FUNCTION "CWA_ScaleRead" : VOID	// FC 42
TITLE = CWA READ SCALE
//
//COPYRIGHT:    (C) 1996 BY  BUHLER LTD.
//                           CH-9240 UZWIL  SWITZERLAND
//
//PRODUCT:      CWA
//
//TITLE:        SCALE CONTROL: READ SCALE
//
//-------------------------------------------------------------------------
//
//IDENT:        AUTOR:              DEPT:                         DATE:
//
//FC42.3.1      A. Egli             CT3                           29-Jun-2004
//              InLocal to disable alarm EsReading
//FC42.3.0      A. Egli             CT3                            8-Feb-2000
//              BCD: Check niybble in range '0' to '9'
//FC42.2A       A. Egli             CT3                           23-Feb-99
//              ERG2: DBX125.7: ParErg2Parallel (16+4Bit)
//              Attention: By Pulse input Bit-Number new on DBB134 not DBB135
//FC42.1D       A. Egli             CT3                           22-Oct-98
//              ERG2: DBX125.6: ParErg2DP
//
//FC42.1C       A. Egli             CT3                           16-Jan-98
//              Fault Reading BCD Value
//
//FC42.1B       A. Egli             CT3                           20-Jan-98
//              Update to  Version S5 2A
//
//FC42.1A       S. Kalberer         AEE61                         24-APR-96
//              1st Release in S7, converted from FB42.1B
//
//-------------------------------------------------------------------------
//
//PURPOSE:      MANUAL : CWAMAN
//
//RESTRICTIONS:
//
//-------------------------------------------------------------------------
//
//
//ACTUAL DB BY CALL: SCALE    DB
//
AUTHOR : EA
FAMILY : CWA
NAME : CWARead
VERSION : 3.1
VAR_TEMP
  AddrPointer : DWORD ;
  tmpValue : DWORD ;
END_VAR
BEGIN
NETWORK
TITLE = BCD/ERG
      AN    DBX 125.1;	// ParERG
      AN    DBX 125.0;	// ParBCD
      JC    NX02;
      A     DBX 57.0;	// inp_ReadingLocked
      O     DBX 125.5;	// ParmeasurmentASW
      JC    NX02;
      A     DBX 125.1;	// ParERG
      JC    ERG;	// === BCD (MINIPOND)==============
      L     DBB 135;	// ParAddrInp2Word
      SLD   3;
      T     #AddrPointer;
      L     DBB 134;	// ParAddrInpBit
      L     PIW [#AddrPointer];	// temp2
      SRW;	// Bit 0= sign
      T     DBW 154;	// --> temp2
      AN    DBX 155.1;	// inp_data_ready
      JC    D_R;
      L     DBW 132;	// ParAddrInp1Word
      SLD   3;
      T     #AddrPointer;
      L     PIW [#AddrPointer];
      T     DBW 152;	// --> temp1
      L     W#16#FFFF;
      ==I;
      JC    ERR1;	// --> reading error
// Begin [3A]  
//    Tesat Digit in range ['0' .. '9']   
      L     DBW 152;	// temp1
      L     W#16#F000;
      AW;
      SRW   12;	// Move to bottom nybble
      L     9;
      >I;
      JC    D_R;	// --> Nibble BCD conversion error
      L     DBW 152;	// temp1
      L     W#16#F00;
      AW;
      L     W#16#900;
      >I;
      JC    D_R;	// --> Nibble BCD conversion error
      L     DBW 152;	// temp1
      L     W#16#F0;
      AW;
      L     W#16#90;
      >I;
      JC    D_R;	// --> Nibble BCD conversion error
      L     DBW 152;	// temp1
      L     W#16#F;
      AW;
      L     W#16#9;
      >I;
      JC    D_R;	// --> Nibble BCD conversion error
// End [3A] 
      L     DBW 152;	// temp1
      BTD;
      AN    DBX 155.2;	// inp_10000
      ON    DBX 124.0;	// ParBCD_Inp10000
      JC    B20;
      +     10000;
B20:  AN    DBX 155.3;	// inp_20000
      ON    DBX 124.1;	// ParBCD_Inp10000
      JC    B40;
      +     L#20000;	// +20000
B40:  AN    DBX 155.4;	// inp_40000
      ON    DBX 124.2;	// ParBCD_Inp10000
      JC    B80;
      +     L#40000;	// +40000
B80:  AN    DBX 155.5;	// inp_80000
      ON    DBX 124.3;	// ParBCD_Inp10000
      JC    BX;
      +     L#80000;	// +80000
BX:   A     DBX 155.0;	// inp_positiv
      JC    POS;
      JU    NEG;	// === ERG ======================
ERG:  L     DBW 132;	// ParAddrInp1Word
      SLD   3;
      T     #AddrPointer;
      L     PIW [#AddrPointer];
      T     DBW 152;	// --> temp1
      AN    DBX 152.6;	// temp1.fault
      JC    ERR1;
      A     DBX 152.7;	// temp1.data_ready
      JC    READ;	// ==== Not data ready ============
D_R:  L     DBW 138;	// ME.VarNotDataReadyCnt
      +     1;
      T     DBW 138;	// --> ME.VarNotDataReadyCnt
      L     DBW 136;
      <I;	// ME.ParNotDataReadyCntMax
      JC    NX02;
      L     77;	// CODE: Time_out Data_ready
ERRO: T     DBW 246;	// --> ErrCodeWorking
      AN    DBX 55.5;	//InLocal      [3.1]
      O     DBX 43.7;	//InfActive    [3.1] 
      S     DBX 244.2;	// --> Fault.EsReading
      JU    NX02;
ERR1: L     78;	// CODE: Fault
      JU    ERRO;
READ: L     W#16#FFF;	// 12-BIT
      AW;
      A     DBX 152.4;	// sign=positiv
      JC    POS;
NEG:  L     0;
      TAK;
      -D;
POS:  T     DBD 152;	// var_temp_1/temp2
      L     DBD 148;	// ME.VarScaleValueInput
      -D;
      L     DBW 130;	// ME.ParDiffReadWtMax
      JP    X2;
      INVI;	// invert
      TAK;
X2:   <=I;
      O     DBX 81.0;	// Loc.Flag.Inf2Reading
      JC    OK;
      S     DBX 81.0;	// Loc.Flag.Inf2Reading
      JU    NX02;
OK:   R     DBX 81.0;	// Loc.Flag.Inf2Reading
      L     DBD 152;	// var_temp_1/temp2
      T     DBD 148;	// ME.VarScaleValueInput
      L     0;
      T     DBW 138;	// --> var_NotDataReadyCnt
NETWORK
TITLE = ERG2
NX02: AN    DBX 125.6;	// ParERG2DP
      AN    DBX 125.7;	// ParERG2Parallel
      JC    e2NX;
      A     DBX 57.0;	// inp_ReadingLocked
      O     DBX 125.5;	// ParmeasurmentASW
      JC    e2NX;
      A     DBX 125.6;	// ParERG2DP
      JC    ERDP;
//ERG2Parallel
      L     DBB 135;	// ParAddrInp2Word
      SLD   3;
      T     #AddrPointer;
      L     DBB 134;	// ME.ParAddrBit
      L     PIW [#AddrPointer];
      SRW;	// Bit 0= sign
      T     #tmpValue;
      SLW   12;
      T     DBW 152;	// --> temp1
      L     DBW 132;	// ParAddrInp1Word
      SLD   3;
      T     #AddrPointer;
      L     PIW [#AddrPointer];
      T     #tmpValue;
      JU    ERD;
//ERG2DP
ERDP: L     DBW 132;	// ParAddrInp1Word
      SLD   3;
      T     #AddrPointer;
      L     PID [#AddrPointer];
      T     #tmpValue;
      SRD   12;
      T     DBW 152;	// --> temp1
ERD:  AN    DBX 152.6;	// temp1.fault
      JC    e2E1;
      A     DBX 152.7;	// temp1.data_ready
      JC    e2RE;	// ==== Not data ready ============
      L     DBW 138;	// ME.VarNotDataReadyCnt
      +     1;
      T     DBW 138;	// --> ME.VarNotDataReadyCnt
      L     DBW 136;
      <I;	// ME.ParNotDataReadyCntMax
      JC    e2NX;
      L     77;	// CODE: Time_out Data_ready
e2EO: T     DBW 246;	// --> ErrCodeWorking
      AN    DBX 55.5;	//InLocal      [3.1]
      O     DBX 43.7;	//InfActive    [3.1] 
      S     DBX 244.2;	// --> Fault.EsReading
      JU    e2NX;
e2E1: L     78;	// CODE: Fault
      JU    e2EO;
e2RE: L     #tmpValue;
      L     DW#16#FFFFFF;	// 24-BIT
      AD;
      A     DBX 152.4;	// sign=positiv
      JC    e2PO;
      NEGD;
e2PO: T     DBD 152;	// var_temp_1/temp2
      L     DBD 148;	// ME.VarScaleValueInput
      -D;
      L     DBW 130;	// ME.ParDiffReadWtMax
      JP    e2X2;
      INVI;	// invert
      TAK;
e2X2: <=I;
      O     DBX 81.0;	// Loc.Flag.Inf2Reading
      JC    e2OK;
      S     DBX 81.0;	// Loc.Flag.Inf2Reading
      JU    e2NX;
e2OK: R     DBX 81.0;	// Loc.Flag.Inf2Reading
      L     DBD 152;	// var_temp_1/temp2
      T     DBD 148;	// ME.VarScaleValueInput
      L     0;
      T     DBW 138;	// --> var_NotDataReadyCnt
NETWORK
TITLE = Impulse
e2NX: AN    DBX 125.2;	// ParPulseInterruptCall
      AN    DBX 125.3;	// ParPulseTimeCall
      JC    NX03;	// 
      A     DBX 57.0;	// ToSSW.InpReadingLocked
      O     DBX 125.5;	// ParMesurmentASW
      JC    NX03;	// 
      A     DBX 125.2;	// ParPulseInterruptCall
      JC    IM_I;
// -- Time CALL -----------------
      L     DBW 132;	// ME.ParAddr1Word
      SLD   3;
      T     #AddrPointer;
      L     DBB 134;	// ME.ParAddrBit  [REL.2A]
      L     PIB [#AddrPointer];
      SRW;	// Bit 0= sign
      T     DBW 154;	// -> Bit 0 = Copy of the Input
      A     DBX 81.1;	// Loc.Flag.InfFlagInpPulse
      ON    DBX 155.0;	// copy of the Input
      JC    OUT;
IM_I: L     DBD 148;	// ME.VarScaleValueInput
      +     L#1;
      T     DBD 148;	// ->ME.VarScaleValueInput
OUT:  A     DBX 155.0;	// copy of the Input
      =     DBX 81.1;	// inf_positive_flag_inp
NETWORK
TITLE = Calulate value absolute
NX03: L     DBD 148;	// ME.VarScaleValueInput
      DTR;
      L     DBD 126;	// Parscale_unit
      *R;
      RND;
      T     DBD 254;	// --> scale_value_absolute
NETWORK
TITLE = Test weight
      L     DBD 254;	// ScaleWt
      L     DBD 140;	// ME.VarCutoffWt
      AN    DBX 7.0;
      JC    POS2;
      TAK;
POS2: <D;
      O     DBX 248.1;	// StaReconveying
      O     DBX 125.4;	// ParDosingRemote
      AN    DBX 252.1;	// StaScrapBatch
      AN    DBX 58.1;	// CmdAbortBatch
      JC    NX05;	// 
      S     DBX 81.2;	// Loc.Flag.InfFlagStopValue
      R     DBX 42.6;	// ToASW.OutpFast
      R     DBX 42.7;	// ToASW.OutpDosing
NETWORK
TITLE =
NX05: BE;
END_FUNCTION

FUNCTION "GCS7_LogConvert" : VOID	// FC 45
TITLE = Log: Message Converter for LOG Entry
//COPYRIGHT:     (C) 1996 BY  BUEHLER LTD. 
//                            CH-9240 UZWIL  SWITZERLAND
//
//PRODUCT:      GCS7 
//
//TITLE:        Message Converter for LOG Entry
//
//--------------------------------------------------------------------------
//
//IDENT:        AUTOR:              DEPT:                       DATE:
//
//FC45.1.2      A. Egli             CT3                         04.03.2003
//              Redesign, M11.2
//FC45.1B       A. Egli             CT3                         26.03.1999
//              Special format for MELE: MsgType>=7000
//FC45.1A       S. Kalberer         AEE61                       27-Sep-1996
//              1st Release in S7, converted from FX251.2A
//
//--------------------------------------------------------------------------
//
//PURPOSE:       DATA-CONVERT FOR PRINTER PER LOG WITH PC
//
//RESTRICTIONS:  S7
//
//--------------------------------------------------------------------------
//
AUTHOR : EA
FAMILY : GCS7LL
NAME : MECONV
VERSION : 0.0
VAR_INPUT
  ObjectNo : INT ;	//Is used for communication with PC
  MsgType : INT ;	//Is used for message translation
  ClassMsgTxt : WORD ;	//Contains MessageClass and MessageTextNumber
  OType : INT ;	//Object Type
END_VAR
VAR_TEMP
  tmpHeader : WORD ;
  tmpPara2 : WORD ;
  tmpObjectNo : WORD ;
  tmpLineNo : WORD ;
  tmpMsgType : WORD ;
  tmpGr : INT ;
  tmpIndex : INT ;
END_VAR
BEGIN
NETWORK
TITLE =  MESSAGE
//Standard GCS90
      L     #ObjectNo;	// Change type INT --> WORD
      T     #tmpObjectNo;
      L     #ClassMsgTxt;	// Load: HighByte= Class ¦ Low Byte= TextNo (8 Bit)
      SRW   8;	// Delete TextNo
      SLW   5;
      +     13;	// add MessageFormatNo
      T     #tmpHeader;	//-> Header=Format := Class ¦ MsgFormatNo
      L     #ClassMsgTxt;	// Load: HighByte= Class ¦ Low Byte= TextNo (8 Bit)
      L     2#11111111;	// Delete Class
      AW;
      L     #MsgType;
      SLW   8;
      OW;
      T     #tmpPara2;	//-->Para2 := MsgType ¦ TextNo
      L     "GCS7_Gr_OutLine";
      T     #tmpLineNo;
      L     #MsgType;
      T     #tmpMsgType;
      A     "GCS7_Gr_OutLogOff";
      JC    EQ00;
      CALL  "SYS_LOG_EntryQueue" (
           DBNumber                 := 5,
           Header                   := #tmpHeader,
           Para1                    := #tmpObjectNo,
           Para2                    := #tmpPara2,
           Para3                    := #tmpLineNo,
           Para4                    := #tmpMsgType,
           Para5                    := W#16#0,
           Para6                    := W#16#0,
           Para7                    := W#16#0,
           Para8                    := W#16#0,
           Para9                    := W#16#0,
           Para10                   := W#16#0,
           Para11                   := W#16#0);	//---Call Message Entry--- /  Queue DB Number                 /  Format /  ObjectNumber /  MsgType ¦ TextNo /  Line /  MsgType S7 /  not used  /  not used  /  not used  /  not used  /  not used  /  not used  /  not used
EQ00: NOP   0;
NETWORK
TITLE = End of Block
END_FUNCTION

FUNCTION "SYS_LOG_EntryQueue" : VOID	// FC 46
TITLE = Log: Message Entry
//COPYRIGHT:    (C) 1996 BY  BUEHLER LTD. 
//                           CH-9240 UZWIL  SWITZERLAND
//
//PRODUCT:      GCS7
//
//TITLE:        Entry in QUEUE for GCS90-Upper-Level
//
//-------------------------------------------------------------------------
//
//IDENT:        AUTHOR:             DEPT:                       DATE:
//
//FC46.2.0      A.Egli              CT3                        14-Jul-2004
//              CmdAddFirst
//FC46.1.1      A.Egli              CT3                        11-Oct-2001
//              Program fault auf Version 1.0 corrected
//FC46.1.0      A.Egli              CT3                        16-Aug-2001
//              Reduce local data
//FC46.1A       S. Kalberer         AEE61                       4-Dec-1996
//              1st Release in S7, converted from FB46.2A
//
//-------------------------------------------------------------------------
//
//PURPOSE:      MANUAL : see [CTRxxMAN]
//              This function entries a print order of 12 DBW (12 WORDS) in
//              in a waiting queue (WQ).
//
//RESTRICTIONS: S7
//              Only for message administration on PC 
//
//INTERRUPT-
// HANDLING:    LOCKED:   SEQUENCE 1
//              RELEASE:  SEQUENCE 4, 5 AND 6
//
//-------------------------------------------------------------------------
//
//        MESSAGE ENTRY               
//   +------------------------+   
// ->¦ DBNumber               ¦           LOG-DB
//   ¦                        ¦       +--------------+
// ->¦ Header                 ¦ ====> ¦  RINGBUFFER  ¦
// ->¦ Para1                  ¦       ¦              ¦
// ->¦ Para2                  ¦       ¦              ¦
// ->¦ Para3                  ¦       +--------------+
// ->¦ Para4                  ¦
// ->¦ Para5                  ¦
// ->¦ Para6                  ¦
// ->¦ Para7                  ¦
// ->¦ Para8                  ¦
// ->¦ Para9                  ¦
// ->¦ Para10                 ¦
// ->¦ Para11                 ¦
//   +------------------------+
//
AUTHOR : EA
FAMILY : GCS7SYS
NAME : MESENTRY
VERSION : 2.0
VAR_INPUT
  DBNumber : INT ;	//Queue DB-Number
  Header : WORD ;	//Header
  Para1 : WORD ;	//Parameter1
  Para2 : WORD ;	//Parameter2
  Para3 : WORD ;	//Parameter3
  Para4 : WORD ;	//Parameter4
  Para5 : WORD ;	//Parameter5
  Para6 : WORD ;	//Parameter6
  Para7 : WORD ;	//Parameter7
  Para8 : WORD ;	//Parameter8
  Para9 : WORD ;	//Parameter9
  Para10 : WORD ;	//Parameter10
  Para11 : WORD ;	//Parameter11
END_VAR
VAR_TEMP
  tmpQueueDB : INT ;
  tmpHeader : WORD ;
  tmpCnt : WORD ;	//temp loop counter
  tmpSourceAddress : DWORD ;	//temp Source Address
  tmpBlockLength : WORD ;	//temp Message BlockLength
  tmpEndOfQueue : INT ;
  tmpOpenDB : INT ;
  tmpBytePrev : INT ;
  tmpMsgActive : BOOL ;
END_VAR
BEGIN
NETWORK
TITLE =  SAVE INPUT 
//---Save Input Parameter into temp variables
      L     #DBNumber;
      T     #tmpQueueDB;
      L     DBNO;
      T     #tmpOpenDB;
      OPN   DB [#tmpQueueDB];
      L     24;
      T     #tmpBlockLength;
//-- Init ---
      L     DBW 8;	// VarNrOfMsgInQueue
      L     0;
      <>I;
      JC    T0;
      L     DBW 2;	// ParDWstartQueue
      T     DBW 10;	// -> varDWwrite
      T     DBW 12;	// -> varDWread
// 
T0:   L     DBW 10;	// varDWwrite
      L     DBW 2;	// ParDWstartQueue
      >I;
      JC    T2;
      T     DBW 10;	// -> varDWwrite
T2:   L     DBW 12;	// varDWread
      L     DBW 2;	// ParDWstartQueue
      >I;
      JC    T3;
      T     DBW 12;	// -> varDWread
T3:   L     DBW 6;	// ParMaxNrOfMsg
      L     #tmpBlockLength;
      *I;
      L     DBW 2;	// ParDWstartQueue
      +I;	// --> Address end of queue
      T     #tmpEndOfQueue;
      L     DBW 6;	// ParMaxNrOfMsg 
NETWORK
TITLE =  PROLOG
      L     DBW 10;	// VarDWWrite 
      L     #tmpBlockLength;	// Block-Length
      +I;
      L     #tmpEndOfQueue;
      >I;
      JC    OUT;	//-->BREAK-OFF   [2.0]
NETWORK
TITLE =  WAITINGQUEUE FULL
//IF WAITINGQUEUE IF FULL
//  THEN
//     BREAK-OFF
      L     DBW 6;	// ParMaxNrOfMsg
      L     DBW 8;	// VarNrOfMsgInQueue
      <=I;	// 
      JC    OUT;	//-->BREAK-OFF   [2.0]
NETWORK
TITLE =  PUT PRINT ORDER IN QUEUE
//IF THERE IS ENOUGH PLACE FOR TWO MESSAGES AT LEAST
//  THEN
//    PUT PRINTORDER INTO WQ
      L     DBW 6;	//ParMaxNrOfMsg
      +     -1;
      L     DBW 8;	//VarNrOfMsgInQueue
      <=I;
      JC    FULL;
      L     DBW 10;	// VarDWWrite 
      SLD   3;	// 
      LAR1;	//--> Write address
NETWORK
TITLE = [2.0] Fast Message
//Immediately Logging at PC Interface
      NOP   0;
//[2.0]--->
      AN    DBX 46.6;	//CmdAddFastMsg
      JC    imJ0;
//When old message was already read by PC then copy 
//the new message also to queue
      A     DBX 57.0;	// HskPLCtoPC
      O     DBX 57.1;	// HskPLCtoPC
      O     DBX 57.2;	// HskPLCtoPC
      O     DBX 57.3;	// HskPLCtoPC
      =     #tmpMsgActive;
      JC    imAC;
      L     1;
      T     "SYS_LOG_Queue".PC.NrOfMessageInQueue;
      JU    imPC;
//Calculate orginal position of message
imAC: L     DBW 8;	//VarNrOfMsgInQueue
      L     0;	// 
      ==I;	// 
      L     DBW 2;	//ParDWstartQueue
      JC    aPrv;	// 
      L     DBW 12;	//varDWread
      L     #tmpBlockLength;	// 
      -I;	// 
      L     DBW 2;	//ParDWstartQueue
      >=I;	// 
      TAK;	// 
      JC    aPrv;	// 
      L     #tmpEndOfQueue;	// 
      L     #tmpBlockLength;	// 
      -I;	// 
aPrv: T     #tmpBytePrev;
      T     DBW 12;	// varDWread
      SLD   3;	// 
      LAR1;	//--> Write address in queue
//When new message was not read then copy message back to queue
//Copy old Message back to Queue
      L     DBD 60;
      T     DBD [AR1,P#0.0];
      L     DBD 64;
      T     DBD [AR1,P#4.0];
      L     DBD 68;
      T     DBD [AR1,P#8.0];
      L     DBD 72;
      T     DBD [AR1,P#12.0];
      L     DBD 76;
      T     DBD [AR1,P#16.0];
      L     DBD 80;
      T     DBD [AR1,P#20.0];
//----Write Message in LOG-queue
imPC: LAR1  P#DBX 60.0;
      OPN   DB [#tmpOpenDB];
      L     #Header;
      OPN   DB [#tmpQueueDB];
      T     DBW [AR1,P#0.0];
      OPN   DB [#tmpOpenDB];
      L     #Para1;
      OPN   DB [#tmpQueueDB];
      T     DBW [AR1,P#2.0];
      OPN   DB [#tmpOpenDB];
      L     #Para2;
      OPN   DB [#tmpQueueDB];
      T     DBW [AR1,P#4.0];
      OPN   DB [#tmpOpenDB];
      L     #Para3;
      OPN   DB [#tmpQueueDB];
      T     DBW [AR1,P#6.0];
      OPN   DB [#tmpOpenDB];
      L     #Para4;
      OPN   DB [#tmpQueueDB];
      T     DBW [AR1,P#8.0];
      OPN   DB [#tmpOpenDB];
      L     #Para5;
      OPN   DB [#tmpQueueDB];
      T     DBW [AR1,P#10.0];
      OPN   DB [#tmpOpenDB];
      L     #Para6;
      OPN   DB [#tmpQueueDB];
      T     DBW [AR1,P#12.0];
      OPN   DB [#tmpOpenDB];
      L     #Para7;
      OPN   DB [#tmpQueueDB];
      T     DBW [AR1,P#14.0];
      OPN   DB [#tmpOpenDB];
      L     #Para8;
      OPN   DB [#tmpQueueDB];
      T     DBW [AR1,P#16.0];
      OPN   DB [#tmpOpenDB];
      L     #Para9;
      OPN   DB [#tmpQueueDB];
      T     DBW [AR1,P#18.0];
      OPN   DB [#tmpOpenDB];
      L     #Para10;
      OPN   DB [#tmpQueueDB];
      T     DBW [AR1,P#20.0];
      OPN   DB [#tmpOpenDB];
      L     #Para11;
      OPN   DB [#tmpQueueDB];
      T     DBW [AR1,P#22.0];
//Set handshake bits
      L     DBW 44;	// ParPCconnection
      SLD   4;
      T     DBW 56;	// HskPLCtoPC
      SET;
      S     DBX 41.0;	//---Set change-bit
//When old message was already read by PC then copy 
//the new message also to queue
      A     #tmpMsgActive;
      JC    L002;
      JU    OUT;
imJ0: NOP   0;
//<---[2.0]
NETWORK
TITLE = Store Message in queue
//----Write Message in LOG-queue
      OPN   DB [#tmpOpenDB];
      L     #Header;
      OPN   DB [#tmpQueueDB];
      T     DBW [AR1,P#0.0];
      OPN   DB [#tmpOpenDB];
      L     #Para1;
      OPN   DB [#tmpQueueDB];
      T     DBW [AR1,P#2.0];
      OPN   DB [#tmpOpenDB];
      L     #Para2;
      OPN   DB [#tmpQueueDB];
      T     DBW [AR1,P#4.0];
      OPN   DB [#tmpOpenDB];
      L     #Para3;
      OPN   DB [#tmpQueueDB];
      T     DBW [AR1,P#6.0];
      OPN   DB [#tmpOpenDB];
      L     #Para4;
      OPN   DB [#tmpQueueDB];
      T     DBW [AR1,P#8.0];
      OPN   DB [#tmpOpenDB];
      L     #Para5;
      OPN   DB [#tmpQueueDB];
      T     DBW [AR1,P#10.0];
      OPN   DB [#tmpOpenDB];
      L     #Para6;
      OPN   DB [#tmpQueueDB];
      T     DBW [AR1,P#12.0];
      OPN   DB [#tmpOpenDB];
      L     #Para7;
      OPN   DB [#tmpQueueDB];
      T     DBW [AR1,P#14.0];
      OPN   DB [#tmpOpenDB];
      L     #Para8;
      OPN   DB [#tmpQueueDB];
      T     DBW [AR1,P#16.0];
      OPN   DB [#tmpOpenDB];
      L     #Para9;
      OPN   DB [#tmpQueueDB];
      T     DBW [AR1,P#18.0];
      OPN   DB [#tmpOpenDB];
      L     #Para10;
      OPN   DB [#tmpQueueDB];
      T     DBW [AR1,P#20.0];
      OPN   DB [#tmpOpenDB];
      L     #Para11;
      OPN   DB [#tmpQueueDB];
      T     DBW [AR1,P#22.0];
      JU    NX06;
NETWORK
TITLE =  SET "WAITING QUEUE FULL"
//IF WAITING QUEUE FULL UNLESS ONE PLACE AND NO ERROR SET
//  THEN
//    SET INTERNAL MESSAGE
//    SET ERROR INPUT
FULL: L     DBW 14;	// ParDWMsgFull
      SLD   3;	// 
      T     #tmpSourceAddress;
      L     DBW 10;	// VarDWWrite 
      SLD   3;	// 
      LAR1;	//--> Write address
      L     #tmpBlockLength;	// SET LOOP-Cnt: BLOCK-Length
      SRW   2;	// /4
COLP: T     #tmpCnt;	//==Blocktransfer: "WQ FULL"
      L     DBD [#tmpSourceAddress];	//  SOURCE
      T     DBD [AR1,P#0.0];
      +AR1  P#4.0;	// Target address
      L     #tmpSourceAddress;	//---INC Source address
      +     L#32;	// + 32 Bit
      T     #tmpSourceAddress;
      L     #tmpCnt;	// LOOP Counter
      LOOP  COLP;	// COPY LOOP 
NETWORK
TITLE =  EPILOG
NX06: L     DBW 10;	// VarDWwrite
      L     #tmpBlockLength;
      +I;
      T     DBW 10;	// --> VarDWWrite
      L     #tmpEndOfQueue;
      <I;
      JC    L002;
      L     DBW 2;	// ParDWStartQueue
      T     DBW 10;	// --> VarDWWrite
L002: L     DBW 8;	// VarNrOfMsgInQueue
      +     1;
      T     DBW 8;	//-->VarNrOfMsgInQueue
OUT:  SET;	//[2.0]
      R     DBX 46.6;	//CmdAddFisrt [2.0]
END_FUNCTION

FUNCTION "SYS_LOG_CtrlQueue" : VOID	// FC 47
TITLE = Log: Read Queue Message
//COPYRIGHT:    (C) 1996 BY  BUEHLER LTD. 
//                           CH-9240 UZWIL  SWITZERLAND
//
//PRODUCT:      GCS7
//
//TITLE:        READ from QUEUE for GCS90-Upper-Level
//
//-------------------------------------------------------------------------
//
//IDENT:        AUTHOR:              DEPT:                       DATE:
//
//FC47.2.0      A.Egli               CT3                         14-Jul-2004
//              CmdAddFisrt
//FC47.1A       S. Kalberer          AEE61                       4-Dec-1996
//              1st Release in S7, converted from FB47.2A
//
//-------------------------------------------------------------------------
//
//PURPOSE:      MANUAL : see [CTRxxMAN]
//              This function reads 1 .. max. 4 print-orders out of the 
//              waiting-queue to set ready at the PC-Interface
//
//RESTRICTIONS: S7
//              Only for message administration on PC
//
//-------------------------------------------------------------------------
//
AUTHOR : EA
FAMILY : GCS7SYS
NAME : MESSFORM
VERSION : 2.0
VAR_INPUT
  DBNumber : INT ;	//Queue DB-Number
END_VAR
VAR_TEMP
  tmpDBNumber : WORD ;	//Input Queue-DB
  tmpCnt : WORD ;	//temp loop counter
  tmpSourceAddress : DWORD ;	//temp Source Address
  tmpDestAddress : DWORD ;	//temp Target Address
  tmpTxtBufferPtr : DWORD ;	//ASA Textbuffer Pointer
  tmpBlockLength : WORD ;	//temp Message BlockLength
  tmpEndOfQueue : INT ;
END_VAR
BEGIN
NETWORK
TITLE =  MESSAGE-FORM
NETWORK
TITLE =  ADDRESS/LENGTH QUEUE
      L     #DBNumber;
      T     #tmpDBNumber;
      OPN   DB [#tmpDBNumber];	//>> CALL QUEUE-DB
      L     24;
      T     #tmpBlockLength;
NETWORK
TITLE =  CONFIGURATION TEST
      AN    DBX 46.7;	// CmdResetLog
      JC    L002;	// 
      R     DBX 46.7;	// CmdResetLog
      L     DBW 2;	// ParDWstartQueue
      T     DBW 10;	// -> varDWwrite
      T     DBW 12;	// -> varDWread
      L     0;	// 
      T     DBW 8;	// VarNrOfMsgInQueue
      T     DBW 56;	// HskPLCtoPC
L002: L     DBW 10;	// varDWwrite
      L     DBW 2;	// ParDWstartQueue
      >I;
      JC    T2;
      T     DBW 10;	// -> varDWwrite
T2:   L     DBW 12;	// varDWread
      L     DBW 2;	// ParDWstartQueue
      >I;
      JC    T3;
      T     DBW 12;	// -> varDWread
T3:   L     DBW 6;	// ParMaxNrOfMsg
      L     #tmpBlockLength;
      *I;
      L     DBW 2;	// ParDWstartQueue
      +I;	// --> Address end of queue
      T     #tmpEndOfQueue;
      L     DBLG;
      >I;
      JC    ERRO;	//-->(ERROR= DB to small)
      L     #tmpEndOfQueue;
      L     #tmpBlockLength;
      -I;
      L     DBW 12;	//  
      <I;	// varDWread
      JC    ERRO;	// -->ERROR= Read Pointer
      JU    NX04;
ERRO: BEU;	// ERROR QUEUE
NETWORK
TITLE =  TEST HANDSHAKE
NX04: L     DBW 44;	//---par_PC_connection[2..1]
      L     DBW 44;	//[2.0]
      SLD   4;	//[2.0]
      OW;	//[2.0]
      L     DBW 56;	// HskPLCtoPC
      AW;
      L     DBW 46;	// inf_control (PC Off-Line)
      INVI;	// Complement 1
      AW;
      T     DBW 56;	// HskPLCtoPC
      A     DBX 49.0;	// HskPC1toPLC.MsgDone
      R     DBX 49.0;	// HskPC1toPLC.MsgDone
      R     DBX 57.0;	// HskPLCtoPC.MsgForPC1
      A     DBX 49.1;	//[2.0] HskPC1toPLC.MsgDone
      R     DBX 49.1;	//[2.0] HskPC1toPLC.MsgDone
      R     DBX 57.4;	//[2.0] HskPLCtoPC.MsgForPC1
      A     DBX 51.0;	// HskPC2toPLC.MsgDone
      R     DBX 51.0;	// HskPC2toPLC.MsgDone
      R     DBX 57.1;	// HskPLCtoPC.MsgForPC2
      A     DBX 51.1;	//[2.0] HskPC2toPLC.MsgDone
      R     DBX 51.1;	//[2.0] HskPC2toPLC.MsgDone
      R     DBX 57.5;	//[2.0] HskPLCtoPC.MsgForPC2
      A     DBX 53.0;	// HskPC3toPLC.MsgDone
      R     DBX 53.0;	// HskPC3toPLC.MsgDone
      R     DBX 57.2;	// HskPLCtoPC.MsgForPC3
      A     DBX 53.1;	//[2.0] HskPC3toPLC.MsgDone
      R     DBX 53.1;	//[2.0] HskPC3toPLC.MsgDone
      R     DBX 57.6;	//[2.0] HskPLCtoPC.MsgForPC3
      A     DBX 55.0;	// HskPC4toPLC.MsgDone
      R     DBX 55.0;	// HskPC4toPLC.MsgDone
      R     DBX 57.3;	// HskPLCtoPC.MsgForPC4
      A     DBX 55.1;	//[2.0] HskPC4toPLC.MsgDone
      R     DBX 55.1;	//[2.0] HskPC4toPLC.MsgDone
      R     DBX 57.7;	//[2.0] HskPLCtoPC.MsgForPC4
      L     0;	//---Handshake is read
      L     DBW 56;	// HskPLCtoPC
      <>I;	// message not read
      BEC;
NETWORK
TITLE =  READ MESSAGE
      L     DBW 8;	// VarNoOfMsgInQueue
      L     0;
      ==I;
      BEC;
      T     DBW 58;	//-->PC.NrOfMessage
      L     P#60.0;	// Address PC.Msg[1]
      T     #tmpTxtBufferPtr;
LOOP: L     DBW 12;	// varDWread 
      SLD   3;
      T     #tmpSourceAddress;
      L     #tmpTxtBufferPtr;
      T     #tmpDestAddress;
//--- Copy one msg to PC interface ----
      L     #tmpBlockLength;
      SRW   2;	// /4
RDLP: T     #tmpCnt;
      L     DBD [#tmpSourceAddress];	//  SOURCE: AEA-ReadPointer
      T     DBD [#tmpDestAddress];	//  TARGET: AEA-WorkingMemory
      L     #tmpSourceAddress;	// INC Source address
      +     L#32;	// + 32 Bit
      T     #tmpSourceAddress;
      L     #tmpDestAddress;	// INC Target address
      +     L#32;	// + 32 Bit
      T     #tmpDestAddress;
      L     #tmpCnt;
      LOOP  RDLP;
//--- End Loop copy ----
//--- Increment address
      L     DBW 58;	// PC.NrOfMessage
      +     1;
      T     DBW 58;	//-->PC.NrOfMessage
      L     DBW 12;	// VarDWread
      L     #tmpBlockLength;
      +D;
      T     DBW 12;	//-->VarDWread
      L     #tmpTxtBufferPtr;	//---TARGET : Msg[n]
      L     #tmpBlockLength;
      SLD   3;
      +D;
      T     #tmpTxtBufferPtr;	// -->TARGET : Msg[n+1]
      L     #tmpEndOfQueue;
      L     DBW 12;	// varDWread
      >I;
      JC    L001;
      L     DBW 2;	// ParDWstartQueue
      T     DBW 12;	//--> varDWread
L001: L     DBW 8;	// VarNrOfMsgInQueue
      +     -1;
      T     DBW 8;	//-->VarNoOrMsgInQueue
      L     DBW 58;	// PC.NoOfMessage
      L     DBW 42;	// ParNrOfMsgMemory
      >=I;
      JC    SEND;
      L     DBW 8;	// VarNoOfMsgInQueue
      L     0;
      >I;
      JC    LOOP;
//---Send to PC -----
SEND: L     DBW 44;	// ParPCconnection
      L     DBW 56;	// HskPLCtoPC
      OW;
      T     DBW 56;	// HskPLCtoPC
      S     DBX 41.0;	//---Set change-bit
END_FUNCTION

FUNCTION "SYS_Copy_DBtoDB" : VOID	// FC 49
TITLE = DB Copy
//
//COPYRIGHT:         (C) 1989 BY  BUEHLER BROTHERS LTD.
//                                CH-9240 UZWIL  SWITZERLAND
//
//PRODUCT:          GCS7
//
//TITLE:            DB COPY 
//
//--------------------------------------------------------------------------
//
//IDENT:            BLOTRA.1A    A.EGLI  AEE61                   16-Jun-96
//                    First release 
//--------------------------------------------------------------------------
//
//PURPOSE   : 
//
//RESTRICTIONS :    S7
//
//---------------------------------------------------------------------------
//
//
AUTHOR : EA
FAMILY : GCS7SYS
NAME : BLOCKTRA
VERSION : 0.0
VAR_INPUT
  DBSource : INT ;	//DB number source DB
  ByteSource : INT ;	//Byte Nr first to copy byte
  DBDest : INT ;	//DB number destination DB
  ByteDest : INT ;	//Byte of first byte in destination DB
  NoOfByte : INT ;	//Number of byte to copy
END_VAR
VAR_OUTPUT
  Fault : BOOL ;	//1=Fault; not posible to copy
END_VAR
VAR_TEMP
  Src : ANY ;
  Dest : ANY ;
  error : INT ;
END_VAR
BEGIN
NETWORK
TITLE =
//                  "DBSource"                              "DBDestination"
//                +-----------+                             +-----------+
//                !           !DBB0                         !           !
//                !           !DBB1          "ByteDest"-->( ! --------- !
//                !           !DBB3                       ( !     !     !
//                !           !                           ( !     !     !
//                !           !           +------------>  ( !     !     !
//"ByteSource"--> ! --------- ! )         !               ( !     !     !
//                !     !     ! )         !               ( !-----------!     
//                !     !     ! )  -------+                 !           !
//                ! "NoOfByte"! )                           !           !
//                !     !     ! )                           !           !
//                !-----------!                             !           !
//                !           !   
NETWORK
TITLE =
      L     W#16#1002;	//S7 word
      T     LW 0;	//->Src.type
      T     LW 10;	//->Dest.type
      L     #NoOfByte;
      T     LW 2;	//->Src.factor
      T     LW 12;	//->Dest.factorr
      L     #DBSource;
      T     LW 4;	//->Src.DB
      L     #DBDest;
      T     LW 14;	//->Dest.DB
      L     #ByteSource;
      SLD   3;
      L     DW#16#84000000;
      OD;
      T     LD 6;	//->Src.BitAddress 
      L     #ByteDest;
      SLD   3;	//->Dest.BitAddress
      L     DW#16#84000000;
      OD;
      T     LD 16;
      CALL  "SIEMENS_BLKMOV" (
           SRCBLK                   := #Src,
           RET_VAL                  := #error,
           DSTBLK                   := #Dest);
      L     #error;
      L     0;
      <>I;
      =     #Fault;
END_FUNCTION

FUNCTION "SYS_Copy_Array_Element" : VOID	// FC 50
TITLE = Copy Array Element
//
//COPYRIGHT:    (C) 2004  BUHLER AG, CH-9240 UZWIL, SWITZERLAND
//
//PRODUCT:      GCS7
//
//TITLE:        Copy Array Element  
//
//--------------------------------------------------------------------------
//
//IDENT:        SYSCopyArray.1.0    A.EGLI  CT3                  16-Apr-04
//                  First release 
//--------------------------------------------------------------------------
//
//PURPOSE   : 
//
//RESTRICTIONS :    S7
//
//---------------------------------------------------------------------------
//
//
//Parameter:
//=========
//
//This function is used to copy an array element to a working memory or back.
//
//----------------------------------------------------------------
//Copying Array[x] to working memory
//-----------------------------------
//Source       : Any Pointer to array
//               Array[Index] from this array is copied to Destination
//Destionation : Any Pointer to working memory. 
//               The structure must be equal as the structure in the array  
//
//Index:         Index of the array element, which you like to copy
//               Range: 1 to n
//
//               NOTE: IF Index is out or range then the
//                     Destionation is cleared 
//----------------------------------------------------------------
//Copying Array[x] to working memory
//-----------------------------------
//Source:        Any Pointer to working memory. 
//               The structure must be equal as the structure in the array  
//Destionation:  Any Pointer to array
//               Array[Index] from this array is copied to Destination
//
//Index:         Index of the array element, which you like to copy
//               Range: 1 to n
//
AUTHOR : EA
FAMILY : GCS7SYS
NAME : ARRAYCOP
VERSION : 1.0
VAR_INPUT
  Source : ANY ;	//Array or Struct
  Destination : ANY ;	//Array or Struct
  Index : INT ;	//Index
END_VAR
VAR_OUTPUT
  Fault : BOOL ;	//1=Fault; not posible to copy
END_VAR
VAR_TEMP
  ByteSource : INT ;	//Byte Nr first to copy byte
  ByteDest : INT ;	//Byte of first byte in destination DB
  LenDest : INT ;	//Number of byte to copy
  LenSource : INT ;
  Dest : ANY ;
  Src : ANY ;
  pointer1 : DINT ;
  pointer2 : DINT ;
  tmpFill : INT ;
  error : INT ;
  ByteCopy : INT ;
END_VAR
BEGIN
NETWORK
TITLE = Copy Pointer for Call of Siemens SFC
      NOP   0;
//----------------------------------------
      L     P##Destination;
      T     #pointer1;
      L     P##Dest;
      T     #pointer2;
      LAR1  #pointer1;
      L     W [AR1,P#0.0];
      LAR1  #pointer2;
      T     W [AR1,P#0.0];
      LAR1  #pointer1;
      L     D [AR1,P#2.0];
      LAR1  #pointer2;
      T     D [AR1,P#2.0];
      LAR1  #pointer1;
      L     D [AR1,P#6.0];
      LAR1  #pointer2;
      T     D [AR1,P#6.0];
//----------------------------------------
      L     P##Source;
      T     #pointer1;
      L     P##Src;
      T     #pointer2;
      LAR1  #pointer1;
      L     W [AR1,P#0.0];
      LAR1  #pointer2;
      T     W [AR1,P#0.0];
      LAR1  #pointer1;
      L     D [AR1,P#2.0];
      LAR1  #pointer2;
      T     D [AR1,P#2.0];
      LAR1  #pointer1;
      L     D [AR1,P#6.0];
      LAR1  #pointer2;
      T     D [AR1,P#6.0];
NETWORK
TITLE = Analyse Data Source
      L     P##Source;
      LAR1;
      L     W [AR1,P#2.0];
      T     #LenSource;
      L     D [AR1,P#6.0];
      L     DW#16#FFFFFF;
      L     D [AR1,P#6.0];
      AD;
      SRD   3;
      T     #ByteSource;
NETWORK
TITLE = Analyse Data Destination
      L     P##Destination;
      LAR1;
      L     W [AR1,P#2.0];
      T     #LenDest;
      L     DW#16#FFFFFF;
      L     D [AR1,P#6.0];
      AD;
      SRD   3;
      T     #ByteDest;
NETWORK
TITLE = Test Fault
      L     #LenSource;
      L     #LenDest;
      <I;
      JC    W1;
//Copy Array[x] to Working Memory
      L     #LenSource;
      L     #LenDest;
      /I;
      L     #Index;
      <I;
      O(;
      L     #Index;
      L     1;
      <I;
      );
      =     #Fault;
      JC    CLEA;
      JU    READ;
//Copy Working Memory to Array[x]
W1:   L     #LenDest;
      L     #LenSource;
      /I;
      L     #Index;
      <I;
      O(;
      L     #Index;
      L     1;
      <I;
      );
      =     #Fault;
      BEC;
      JU    WRIT;
NETWORK
TITLE = Copy Array[x] to Working memory
READ: NOP   0;
//---------------------------------------------
//Calculate Nr Byte Source
      L     #Index;
      +     -1;
      L     #LenDest;
      *I;
      L     #ByteSource;	//Input
      +I;
      T     #ByteCopy;
//---------------------------------------------
//Modify pointer Source
      L     P##Src;
      LAR1;
      L     #LenDest;
      T     W [AR1,P#2.0];	//-->Length in Byte
      L     DW#16#FF000000;
      L     D [AR1,P#6.0];
      AD;
      L     #ByteCopy;
      SLD   3;
      OD;
      T     D [AR1,P#6.0];	//-->Bit Nr Source
//---------------------------------------------
//Copy Data
COP1: CALL  "SIEMENS_BLKMOV" (
           SRCBLK                   := #Src,
           RET_VAL                  := #error,
           DSTBLK                   := #Dest);
      L     #error;
      L     0;
      <>I;
      =     #Fault;
      BEU;
NETWORK
TITLE = Copy Working memory to Array[x] 
WRIT: NOP   0;
//---------------------------------------------
//Calculate Nr Byte Source
      L     #Index;
      +     -1;
      L     #LenSource;
      *I;
      L     #ByteDest;
      +I;
      T     #ByteCopy;
//---------------------------------------------
//Modify pointer Destination
      L     P##Dest;
      LAR1;
      L     #LenSource;
      T     W [AR1,P#2.0];	//-->Length in Byte
      L     DW#16#FF000000;
      L     D [AR1,P#6.0];
      AD;
      L     #ByteCopy;
      SLD   3;
      OD;
      T     D [AR1,P#6.0];	//-->Bit Nr Destination
//---------------------------------------------
//Copy Data
      JU    COP1;
NETWORK
TITLE = Clear Destination
      BEU;
CLEA: L     #LenDest;
      L     #LenSource;
      >I;
      BEC;
      L     0;
      T     #tmpFill;
      CALL  "SIEMENS_FILL" (
           BVAL                     := #tmpFill,
           RET_VAL                  := #error,
           BLK                      := #Dest);
END_FUNCTION

FUNCTION "SYS_DeleteDB" : VOID	// FC 51
TITLE = DB Clear
//
//COPYRIGHT:         (C) 1999 BY  BUEHLER AG
//                                CH-9240 UZWIL  SWITZERLAND
//
//PRODUCT:          GCS7
//
//TITLE:            DB CLEAR S7
//
//--------------------------------------------------------------------------
//
//IDENT:            CLEAR.1A    R.STEIGER SC41                     22-Jan-98
//                    First release 
//--------------------------------------------------------------------------
//
//PURPOSE   : 
//
//RESTRICTIONS :    S7
//
//---------------------------------------------------------------------------
//
//
AUTHOR : EA
FAMILY : GCS7SYS
NAME : CLEAR
VERSION : 0.0
VAR_INPUT
  DBDest : INT ;	//DB number destination DB
  ByteDest : INT ;	//Byte of first byte in destination DB
  NoOfByte : INT ;	//Number of byte to delete
END_VAR
VAR_OUTPUT
  Fault : BOOL ;	//1=Fault; not posible to delete
END_VAR
VAR_TEMP
  Src : BYTE ;
  Dest : ANY ;
  error : INT ;
END_VAR
BEGIN
NETWORK
TITLE =
      L     0;
      T     #Src;	//->Source
      L     W#16#1002;	//S7 word
      T     LW 2;	//->Dest.type
      L     #NoOfByte;
      T     LW 4;	//->Dest.factor
      L     #DBDest;
      T     LW 6;	//->Dest.DB
      L     #ByteDest;
      SLD   3;	//->Dest.BitAddress
      L     DW#16#84000000;
      OD;
      T     LD 8;
      CALL  "SIEMENS_FILL" (
           BVAL                     := #Src,
           RET_VAL                  := #error,
           BLK                      := #Dest);	// Source
      L     #error;
      L     0;
      <>I;
      =     #Fault;
END_FUNCTION

FUNCTION "SYS_InitFlagTimer" : VOID	// FC 52
TITLE = TimerFlag
//  
//COPYRIGHT:    (C) 1996  BUHLER AG, CH-9240 UZWIL, SWITZERLAND
//
//PRODUCT:      BASIS
//
//TITLE:        TimerFlag/Scanner
//
//-------------------------------------------------------------------------
//
//IDENT:        AUTHOR:             DEPT:                       DATE:
//
//FC52.2.1      A. Egli             CT3                         26-Oct-2003
//              M3.6: Sys_Tick100msFromFastOB for long scan time
//              M3.7: Sys_Tick200msFromFastOB for long scan time
//              Modifcation OB35 see below
//FC52.2.0      S. Kalberer         CT3                         14-Apr-2000
//              New M10.2: 100ms tick
//FC52.1C       A.Egli              CT3                         13-Aug-1999
//              M9.4: 1s High /1s low  M9.3 0.5s high/0.5s low
//FC52.1B       A.Egli              CT3                         26-NOV-1998
//              1 min Takt
//FC52.1A       S. Kalberer         AEE61                       12-JUN-1996
//              1st Release in S7, converted from FB100.1A
//
//-------------------------------------------------------------------------
//
//PURPOSE:      - make scan A,B,C  (MB3)
//              - make time flags  (MB4,MB5, MB6, MB7)
//              - make flags M9.0-M 9.5
//              - make ticks M11.2-M11.6
//              - init timer group M11.3-M11.5
//
//RESTRICTIONS: Needs CPU-Tactflag-Byte MB 2
//              Needs Z0                          
//                   
//-------------------------------------------------------------------------
//
//
//
//-------------------------
//Code in fast OB: e.g 20ms
//--------------------------
//For CPU with long scan time (>100ms) you must add the following code to a fast 
//OB.
//      U     "Sys.Pulse100ms"            // 10 Hz CPU-Tactmerker
//      FP    "Sys.CPulse100ms"           // Positive rise
//      S     "Sys.Tick100msFromFastOB"   // Sys.Tick100msFromFastOB
//
//      U     "Sys.Pulse200ms"            // 5 Hz CPU-Tactmerker
//      FP    "Sys.CPulse200ms"           // Positive rise
//      S     "Sys.Tick200msFromFastOB"   // Sys.Tick200msFromFastOB
//
//or
//      U     M      2.0                  // 10 Hz CPU-Tactmerker
//      FP    M      1.0                  // Positive rise
//      S     M      3.6                  // Sys.Tick100msFromFastOB 
//
//      U     M      2.1                  // 5 Hz CPU-Tactmerker
//      FP    M      1.1                  // Positive rise
//      S     M      3.7                  // Sys.Tick200msFromFastOB 
//
//
//
//
//
//
AUTHOR : EA
FAMILY : GCS90SYS
NAME : BLINK
VERSION : 2.1
BEGIN
NETWORK
TITLE = Init flags
      CLR;
      =     "SYS_infLog0";	// "LOW"-MERKER
      SET;
      =     "SYS_infLog1";	// "HIGH"-MERKER
// Clear flags
      R     "SYS_Scan0_Tick100ms";	// [2.0] Scan0.Tick100ms
      R     "SYS_Scan0_Tick200ms";	// Scan0.Tick200ms
      R     "SYS_Scan0_Tick500ms";	// Scan0.Tick500ms
      R     "SYS_Scan0_Tick1s";	// Scan0.Tick1s
      R     "SYS_Scan0_Tick1min";	// Scan0.Tick1min
// Flasher
      AN    "SYS_CycleFlasher";	// Toggle
      =     "SYS_CycleFlasher";	// Toggle
      A     "CPU_Pulse1000ms";	// 1Hz CPU-Tact
      =     "SYS_Pulse500ms";	// Flasch500ms
      A     "CPU_Pulse2000ms";	// 1Hz CPU-Tact
      =     "SYS_Pulse1000ms";	// Flasch1s
NETWORK
TITLE = Scan
      A     "SYS_ScanA_IsOn";	// ScanA
      JC    SCA;
      A     "SYS_ScanB_IsOn";	// ScanB
      JC    SCB;
      A     "SYS_ScanC_IsOn";	// ScanB
      JC    SCC;
SCA:  R     "SYS_ScanA_IsOn";	// ScanA
      S     "SYS_ScanB_IsOn";	// ScanB
      R     "SYS_ScanA_Tick200ms";	// TickA_200ms
      R     "SYS_ScanA_Tick500ms";	// TickA_500ms
      R     "SYS_ScanA_Tick1s";	// TickA_1s
      R     "SYS_ScanA_Tick1min";	// TickA_1min
      JU    TIME;
SCB:  R     "SYS_ScanB_IsOn";	// ScanB
      S     "SYS_ScanC_IsOn";	// ScanC
      R     "SYS_ScanB_Tick200ms";	// TickB_200ms
      R     "SYS_ScanB_Tick500ms";	// TickB_500ms
      R     "SYS_ScanB_Tick1s";	// TickB_1s
      R     "SYS_ScanB_Tick1min";	// TickB_1min
      JU    TIME;
SCC:  R     "SYS_ScanC_IsOn";	// ScanC
      S     "SYS_ScanA_IsOn";	// ScanA
      R     "SYS_ScanC_Tick200ms";	// TickA_200ms
      R     "SYS_ScanC_Tick500ms";	// TickA_500ms
      R     "SYS_ScanC_Tick1s";	// TickA_1s
      R     "SYS_ScanC_Tick1min";	// TickA_1min
NETWORK
TITLE = Tick
// [2.0] 100ms tick
TIME: A     "CPU_Pulse100ms";	// 10 Hz CPU-Tactflag
      FP    "CPU_CopyPulse100ms";	// Positive rise
      O     "Sys_Tick100msFromFastOB";	//[2.1]
      R     "Sys_Tick100msFromFastOB";	//[2.1]
      S     "SYS_Scan0_Tick100ms";	// Tick0_100ms
// 200ms tick
      A     "CPU_Pulse200ms";	// 5 Hz CPU-Tactmerker
      FP    "CPU_CopyPulse200ms";	// Positive rise
      O     "Sys_Tick200msFromFastOB";	//[2.1]
      R     "Sys_Tick200msFromFastOB";	//[2.1]
      S     "SYS_Scan0_Tick200ms";	// Tick0_200ms
      S     "SYS_ScanA_Tick200ms";	// TickA_200ms
      S     "SYS_ScanB_Tick200ms";	// TickB_200ms
      S     "SYS_ScanC_Tick200ms";	// TickC_200ms
// 500ms tick
      A     "CPU_Pulse500ms";	// 2 Hz CPU-Tactmerker
      FP    "CPU_CopyPulse500ms";	// Positive rise
      S     "SYS_Scan0_Tick500ms";	// Tick0_500ms
      S     "SYS_ScanA_Tick500ms";	// TickA_500ms
      S     "SYS_ScanB_Tick500ms";	// TickB_500ms
      S     "SYS_ScanC_Tick500ms";	// TickC_500ms
// 1ms tick
      A     "CPU_Pulse1000ms";	// 1 Hz CPU-Tactmerker
      FP    "CPU_CopyPulse1000ms";	// Positive rise
      S     "SYS_Scan0_Tick1s";	// Tick0_500ms
      S     "SYS_ScanA_Tick1s";	// TickA_500ms
      S     "SYS_ScanB_Tick1s";	// TickB_500ms
      S     "SYS_ScanC_Tick1s";	// TickC_500ms
// 1min tick
      A     "SYS_Scan0_Tick1s";	// Tick0_500ms
      CD    C 0;
      AN    C 0;
      S     "SYS_Scan0_Tick1min";	// Tick0_1min
      S     "SYS_ScanA_Tick1min";	// TickA_1min
      S     "SYS_ScanB_Tick1min";	// TickB_1min
      S     "SYS_ScanC_Tick1min";	// TickC_1min
      L     C#60;
      S     C 0;
NETWORK
TITLE = Out Flag group
// [2.0] 100ms tick
      A     "SYS_Scan0_Tick100ms";	// Tick0_100ms
      =     "GCS7_Gr_OutTick100ms";	// OutTick100ms
// 200ms tick
      A     "SYS_Scan0_Tick200ms";	// Tick0_200ms
      =     "GCS7_Gr_OutTick200ms";	// OutTick200ms
// 500ms tick
      A     "SYS_Scan0_Tick500ms";	// Tick0_500ms
      =     "GCS7_Gr_OutTick500ms";	// OutTick500ms
// 1ms tick
      A     "SYS_Scan0_Tick1s";	// Tick0_1s
      =     "GCS7_Gr_OutTick1s";	// OutTick1s
      =     "SYS_Tick1s";	// Tick1S
// 1min tick
      A     "SYS_Scan0_Tick1min";	// Scan0.Tick1min
      =     "GCS7_Gr_OutTick1min";	// Gr.OutTick1min
END_FUNCTION

FUNCTION "SYS_BitAddress" : VOID	// FC 53
TITLE = Copy Array Element
//
//COPYRIGHT:    (C) 2004  BUHLER AG, CH-9240 UZWIL, SWITZERLAND
//
//PRODUCT:      GCS7
//
//TITLE:        Get Bit Address of any symbol 
//
//--------------------------------------------------------------------------
//
//IDENT:        SYSBitAddr.1.0    A.EGLI  CT3                  10-June-05
//                  First release 
//--------------------------------------------------------------------------
//
//PURPOSE   : 
//
//RESTRICTIONS :    S7
//
//---------------------------------------------------------------------------
//
//
//Parameter:
//=========
//
//This function is used to copy an array element to a working memory or back.
//
//----------------------------------------------------------------
//Copying Array[x] to working memory
//-----------------------------------
//Source       : Any Pointer to array
//               Array[Index] from this array is copied to Destination
//Destionation : Any Pointer to working memory. 
//               The structure must be equal as the structure in the array  
//
//Index:         Index of the array element, which you like to copy
//               Range: 1 to n
//
//               NOTE: IF Index is out or range then the
//                     Destionation is cleared 
//----------------------------------------------------------------
//Copying Array[x] to working memory
//-----------------------------------
//Source:        Any Pointer to working memory. 
//               The structure must be equal as the structure in the array  
//Destionation:  Any Pointer to array
//               Array[Index] from this array is copied to Destination
//
//Index:         Index of the array element, which you like to copy
//               Range: 1 to n
//
AUTHOR : EA
FAMILY : GCS7SYS
NAME : BITADDR
VERSION : 1.0
VAR_INPUT
  Source : POINTER ;	//Array or Struct
END_VAR
VAR_OUTPUT
  OutBitAddr : DWORD ;
END_VAR
BEGIN
NETWORK
TITLE = Analyse Data Source Address
      L     P##Source;
      LAR1;
      L     D [AR1,P#2.0];
      T     #OutBitAddr;
END_FUNCTION

FUNCTION "GCS7_LineCtrlMain" : VOID	// FC 58
TITLE = LineMain
//COPYRIGHT:    (C) 1994 BY  BUHLER AG,CH-9240 UZWIL  SWITZERLAND
//
//PRODUCT:      GCS7
//
//TITLE:        LINE/Job: Main program
//
//-------------------------------------------------------------------------
//
//IDENT:        AUTOR:              DEPT:                         DATE:
//FC58.2.1      A.Egli              CT3                           28-Feb-2006
//              Method 2: Remove nonsense bit DBX  152.0
//FC58.2.0      A.Egli              CT3                            4-Okt-2002
//              New Release with new addresse
//FC58.1.4      A.Egli              CT3                            5-Jul-2000
//              Read command from PC only with F_Define 
//FC58.1.3      A.Egli              CT3                           14-Apr-2000
//              Test Job allready active
//FC58.1C       A.Egli              AEE61                         14-Jan-98
//              Line-Number DBW2
//FC58.1B       A.Egli              AEE61                         14-Jan-98
//               Update  S5 Version 1E
//FC58.1A       A.Egli              AEE61                         18-Jun-96
//               Convert S5--> S7 Version 1D
//
//-------------------------------------------------------------------------
//
//PURPOSE:      MANUAL : GCSOSMAN
//
//RESTRICTIONS:
//
//-------------------------------------------------------------------------
//
//
//FX-PARAMETER:
//------------
//  CODE: CODE of the methode
//        KF +1    : Methode Init     (Communication)
//        KF +2    : Methode Control  (Communication)
//        KF +10   : Methode Commands      (Line)
//        KF +13   : Methode Step          (Line)
//        KF +16   : Methode Summary Mask  (Line)
//
//ACTUAL DB BY CALL: Line-DB
//
//Internal restriction:
//DB : Line-DB
//DI : Section DB
//
//$EJECT
//
//
AUTHOR : EA
FAMILY : GCS7UL
NAME : LineMain
VERSION : 2.1
VAR_INPUT
  CODE : INT ;	// CODE
END_VAR
VAR_TEMP
  VarAdr : DWORD ;
  VarActive : BOOL ;
  VarStopped : BOOL ;
  VarReadyNext : BOOL ;
END_VAR
BEGIN
NETWORK
TITLE =
NETWORK
TITLE =  Methode Init (Communication)
      L     #CODE;
      L     1;
      <>I;
      JC    BEnd;	// 
      L     DBW 144;	// JobWrite.Hsk
      L     0;	// 
      ==I;	// 
      BEC;	// -->no new datas
//==New Data ========================================
      T     DBW 138;	// ->JobRead.ErrElement
      T     DBW 140;	//  ->JobRead.ErrCode
      T     DBW 142;	//  ->JobRead.ErrObject
//==Test job allready active=========================
      L     0;	//  
      L     DBW 154;	// JobWrite.SectionDest
      ==I;	//  
      A(;	//  
      A     DBX 145.0;	//  JobWrite.Hsk.F_Define
      O     DBX 145.1;	// JobWrite.Hsk.F_Execute
      );	// 
      JC    BEr1;	// 
      R     DBX 39.0;	// <--err_job_active      [1.3]
      CALL  "GCS7_SecCtrlSub" (
           CODE                     := 5);	// Soubroutine Search Job /  
      AN    DBX 145.0;	// JobWrite.Hsk.F_Define
      AN    DBX 145.1;	// JobWrite.Hsk.F_Execute
      JC    BEnd;	// --- target section free ?? ----
      A     DBX 39.0;	// <--err_job_active      [1.3]
      L     13;	// error: job all ready active  [1.3]
      JC    BErO;	// 
//==Marke all address section =========================
      L     DBW 154;	//  JobWrite.SectionDest
      T     DBW 20;	// 
      L     0;	// 
      T     DBW 22;	// search_mode section_nr
      CALL  "GCS7_SecCtrlSub" (
           CODE                     := 4);	// Subroutine Search section  /  
      L     DBW 22;	// VarSecDB
      L     0;	// 
      ==I;	// 
      JC    BEr1;	// ->illegal section-nr
      OPN   DI [DBW 22];	//>>>  Call section-DB
      A     DIX 45.7;	// ToASW.InfDataReady
      JC    BEr2;	// ->section_not_ready
      BEU;	// 
//==Error handling ==================================
BEr1: L     10;	// error: illegal section
      JU    BErO;	// 
BEr2: L     11;	// error: section not ready
BErO: T     DBW 140;	// ->JobRead.ErrCode
      L     DBW 154;	//  -> JobWrite.SectionDest
      T     DBW 142;	// ->.JobRead.ErrObject
      L     0;	// 
      T     DBW 144;	// ->JobWrite.Hsk
      S     DBX 41.2;	// ->ChangeBit.CBit3 (interface_free)
      BEU;
BEnd: NOP   0;
NETWORK
TITLE =  Methode Control (Communication)
      L     #CODE;	// 
      L     2;	// 
      <>I;	// 
      JC    CEnd;	// 
      L     DBW 144;	// JobWrite.Hsk
      L     0;	// 
      ==I;	// 
      BEC;	// 
//========== New Data ========================================
      L     DBW 140;	//  err_code
      <>I;	//  
      JC    CINI;	//  
//[2.1]  U     DBX  152.0
      L     DBD 146;	//  JobWrite.ObjMask[1..32]
      L     DBD 150;	//  JobWrite.ObjMask[33..64]
      OD;
      JZ    CINI;	//  --> OK
//===Serach object number which is not answered  =============
      L     1;	//   
      T     DBW 142;	//  -->err_object
      L     P#146.0;	//  JobWrite.ObjMask[1]
CLop: T     #VarAdr;	//   
      A     DBX [#VarAdr];	//  JobWrite.ObjMask[x] 
      JC    Cerr;
      L     DBW 142;	//  JobRead.ErrObject
      +     1;
      T     DBW 142;	//  JobRead.ErrObject
      L     #VarAdr;	//   
      +     1;	//  increment x
      JU    CLop;
//==Error handling ==================================
Cerr: L     20;	//  error: illegal object
      T     DBW 140;	// ->JobRead.ErrCode
CINI: L     0;	//  
      T     DBW 144;	// ->JobWrite.Hsk
      SET;	//  
      S     DBX 41.2;	// ->ChangeBit.CBit3 (interface_free)
      BEU;
CEnd: NOP   0;
NETWORK
TITLE =  Methode commands (Line)
      L     #CODE;
      L     10;
      <>I;
      JC    Dend;
      L     0;	//   
      L     DBD 66;	// ToSSW.Func
      ==D;	//  
      BEC;	//  
      T     DBD 32;	// VarTem[7..8]
      CALL  "GCS7_LineCtrlSub" (
           CODE                     := 3);	// Soubroutine send
      L     0;	//  
      T     DBD 66;	// ToSSW.Func
      BEU;
Dend: NOP   0;
NETWORK
TITLE =  Methode PC_Direct Control (Diagnose)
      L     #CODE;
      L     12;
      <>I;
      JC    Eend;
      OPN   DI 3;	// Change DB and DI
      L     0;	// 
      L     DIW 42;	// DB3.PC.Hsk
      ==I;	// 
      BEC;	// 
//----- Compare Object ID  --------------
      L     DIW 48;	// ) DB3.PC.ObjectType
      L     5000;	// )
      <>I;	// )
      BEC;	// )
      L     DIW 50;	// ) DB3.PC.ObjectNo
      L     DBW 2;	// ) Para.ParLineNr
      <>I;	// )
      BEC;	// )
//----- commands -------------------------
      AN    DIX 43.0;	// PC.Hsk.FDefineCmd
      JC    EdfP;	// 
      L     DID 52;	// DB3.PC.Cmd1
      L     DBD 66;	// ToSSW.Func
      OD;	//  
      T     DBD 66;	// -->ToSSW.Func 
//----- Parameter -------------------------
EdfP: AN    DIX 43.1;	// DB3.PC.Hsk.FDefinePara
      JC    Eexa;	// 
      L     DID 58;	// DB3.PC.Value[1..2]
      T     DBD 90;	// PCWrite.Value1..2 
      L     DID 62;	// DB3.PC.Value[3..4]
      T     DBD 94;	// PCWrite.Value3..4
      L     DID 66;	// DB3.PC.Value[5..6]
      T     DBD 98;	// PCWrite.Value5..6 
Eexa: AN    DIX 43.3;	// DB3.PC.Hsk.FExamine
      JC    Edon;	//  
      L     DBD 90;	// PCWrite.Value1..2 
      T     DID 58;	// DB3.PC.Value[1..2]
      L     DBD 94;	// PCWrite.Value3..4
      T     DID 62;	// DB3.PC.Value[3..4]
      L     DBD 98;	// PCWrite.Value5..6 
      T     DID 66;	// DB3.PC.Value[5..6]
Edon: L     0;
      T     "SYS_DirectCtrlDB".PC.Hsk;	// DB3.PC.Hsk
      T     "SYS_DirectCtrlDB".PC.ErrCode;	// DB3.PC.ErrCode
      SET;	// 
      S     "SYS_DirectCtrlDB".ChangeBit.CBit1;	// -> DB3.ChangeBit.CBit1
      BEU;
Eend: NOP   0;
NETWORK
TITLE =  Methode Step (Line)
      L     #CODE;
      L     13;
      <>I;
      JC    Fend;
      R     #VarActive;
      R     #VarReadyNext;
      S     #VarStopped;
      OPN   DI [DBW 4];	// -->CALL SECTION-DB["LineDB".Para.ParFirstSecDB]
//===read section information===
FLop: A     DIX 45.7;	// "SecDB1".ToASW.InfDataReady
      S     #VarActive;	// ->VarActive
      AN    DIX 111.0;	// "SecDB1".PCRead.Step.StPassive
      R     #VarStopped;	// -> var_stopped
      L     DIW 70;	// "SecDB1".ToSSW.InPrevSecDB
      L     0;	// 
      ==I;	// 
      AN    DIX 45.7;	// "SecDB1".ToASW.InfDataReady
      S     #VarReadyNext;	// ->var_ready
      L     DIW 8;	// "SecDB1".Para.ParNextSecDB
      ==I;	// 
      JC    Fsta;	// -->start
      OPN   DI [DIW 8];	// ->CALL SECTION-DB["SecDB1".Para.ParNextSecDB]
      JU    FLop;	// 
// ===== State-Event ==========
      A     DBX 111.0;
Fsta: A     DBX 111.0;	//  "LineDB1".PCRead.Step. ST_PASSIVE
      JC    FS0;
      A     DBX 111.2;	//  "LineDB1".PCRead.Step.StActive
      JC    FS1;
      A     DBX 111.3;	// "LineDB1".PCRead.Step.StActiveReady
      JC    FS2;
      A     DBX 111.6;	// "LineDB1".PCRead.Step.StIdling
      JC    FS3;
      S     DBX 111.0;	//"LineDB1".PCRead.Step.StPassive
// === ST_PASSIVE  ============
FS0:  A     #VarActive;
      JC    FT01;	// --> StActive
      JU    Fend;
FT01: L     2#100;	// --> StActive
      JU    FTRA;
// === StActive   ============
FS1:  AN    #VarActive;
      JC    FT13;	// --> StIdling
      A     #VarReadyNext;
      JC    FT12;	// --> StActiveReady
      JU    Fend;
FT12: L     2#1000;	// --> StActiveReady
      JU    FTRA;
FT13: L     2#1000000;	// --> StIdling
      JU    FTRA;
// === StActiveReady =======
FS2:  AN    #VarActive;
      JC    FT23;	// --> StIdling
      AN    #VarReadyNext;
      JC    FT21;	// --> StActiveReady
      JU    Fend;
FT21: L     2#100;	// --> StActive
      JU    FTRA;
FT23: L     2#1000000;	// --> StIdling
      JU    FTRA;
// ==== StIdling ==============
FS3:  A     #VarStopped;
      JC    FT30;	// --> StPassive
      A     #VarActive;
      JC    FT31;	// --> StActive
      JU    Fend;	// 
FT30: L     2#1;	// --> StPassive
      JU    FTRA;
FT31: L     2#100;	// --> StActive
// ==== ALL TRANSITION ========
FTRA: T     DBB 111;	// --> "LineDB1".PCRead.Step
      A     "SYS_infLog1";	// 
      S     DBX 41.0;	//"LineDB1".ChangeBit.CBit1
      BEU;
//END:
Fend: NOP   0;
NETWORK
TITLE =  Methode Summary Mask (Line)
      L     #CODE;
      L     16;
      <>I;
      JC    GEnd;
      L     0;
      T     DBD 32;	//  VarFault  = "LineDB1".VarTemp[7,8]
      T     DBD 36;	//  VarStatus = "LineDB1".VarTemp[9,10]
      OPN   DI [DBW 4];	// -->CALL SECTION-DB[Para.ParFirstSecDB]
//Read section Data
GLop: L     DID 114;	//  "SecDB1".PCRead.Fault
      L     DBD 32;	//  VarFault
      OD;	//  
      T     DBD 32;	//  VarFault
      L     DID 118;	//  "SecDB1".PCRead.Status
      L     DBD 36;	//  VarStatus
      OD;	//  
      T     DBD 36;	//  VarStatus
//-- Next section --
      L     0;	// 
      L     DIW 8;	// "SecDB1".Para.ParNextSecDB
      ==I;	// 
      JC    GJ1;	//    
      OPN   DI [DIW 8];	// ->CALL SECTION-DB["SecDB1".Para.ParNextSecDB]
      JU    GLop;	// 
//Store Data
GJ1:  L     DBD 32;	//  VarFault  = "LineDB1".VarTemp[7,8]
      T     DBD 114;	//  "SecDB1".PCRead.Fault
      L     DBD 36;	//  VarStatus = "LineDB1".VarTemp[9,10]
      T     DBD 118;	//  "SecDB1".PCRead.Status
      BEU;
GEnd: NOP   0;
NETWORK
TITLE =  Methode O_LINE
      L     #CODE;	// 
      L     17;	// 
      <>I;	// 
      JC    HEnd;	// 
      L     DBW 82;	// "LineDB1".PCWrite.Hsk
      L     0;	//  
      ==I;	//  
      BEC;
// -- commands --------------
      S     DBX 41.0;	// "LineDB1".ChangeBit.CBit1 (new data)
      S     DBX 41.1;	// "LineDB1".ChangeBit.CBit2 (interface free)
      L     0;	// 
      L     DBD 86;	//"LineDB1".PCWrite.Func
      ==D;	// 
      ON    DBX 83.0;	// "LineDB1".PCWrite.Hsk.F_Define
      JC    HIni;	// 
      T     DBD 32;	// VarFunction =  "LineDB1".VarTemp[7,8]
      CALL  "GCS7_LineCtrlSub" (
           CODE                     := 3);	// Soubroutien send commands
//Line:Extended command  
      L     DBW 90;	// "LineDB".PCWrite.ExtFuncOn
      L     DBW 126;	// "LineDB".PCRead.ExtStatus
      OW;
      T     DBW 126;	// "LineDB".PCRead.ExtStatus
      L     DBW 92;	// "LineDB".PCWrite.ExtFuncOff
      INVI;
      L     DBW 126;	// "LineDB".PCRead.ExtStatus
      AW;
      T     DBW 126;	// "LineDB".PCRead.ExtStatus
HIni: L     0;	// 
      T     DBW 82;	// "LineDB1".PCWrite.Hsk
      BEU;
HEnd: NOP   0;
NETWORK
TITLE =
END_FUNCTION

FUNCTION "GCS7_LineCtrlSub" : VOID	// FC 59
TITLE = Subroutine Line
//COPYRIGHT:    (C) 1994 BY  BUHLER LTD.
//                           CH-9240 UZWIL  SWITZERLAND
//
//PRODUCT:      GCS7
//
//TITLE:        COMMUNICATION/LINE: SUBROUTINE
//
//-------------------------------------------------------------------------
//
//IDENT:        AUTOR:              DEPT:                         DATE:
//
//FB59.2.0      A.Egli              CT3                           04-Okt-2002
//              New release with new address
//FB59.1.0      A.Egli              AEE6                          19-Jun-96
//              Convert from S5 to S7 (Version 1B)
//-------------------------------------------------------------------------
//
//PURPOSE:      MANUAL : GCSOSMAN
//
//RESTRICTIONS:
//
//-------------------------------------------------------------------------
//
//Input Parameter:
//=========================
//- Code: Called Function 
//   1 =Subroutine "Object Address"
//   2 =Subroutine "Reset ObjMask "
//   3 =Subroutine "Send Command"
//
//
//
AUTHOR : EA
FAMILY : GCS7UL
NAME : COM_SUBR
VERSION : 2.0
VAR_INPUT
  CODE : INT ;	// CODE
END_VAR
VAR_TEMP
  VarAdrBit : DWORD ;
  VarCountLoop : INT ;
  VarBitAdrRead : DWORD ;
END_VAR
BEGIN
NETWORK
TITLE =
NETWORK
TITLE =  Code 1: Subroutine: Object Address
// Suche Zeiger auf Variable Solldatenblock des Objektes n
// Search the pointer to the data-block of objekt n
//
// CALL by methode decoder
// INPUT  : ACTUAL DB BY CALL =LineDB
// INPUT  : LineDB.VarTemp[1] DBW20: ObjectNr
//
// OUTPUT : LineDB.VarTemp[2] DBW22: First DW OF THE ACTUAL BLOCK
//          SPECIAL DBW22=0 : no data block
      L     #CODE;
      L     1;
      <>I;
      JC    END;
      L     DBW 22;
      L     0;	//  
      T     DBW 22;	// -->"LineDB1".VarTemp[2]= VarDWNr
      L     DBW 20;	// LineDB.VarTemp[1] = ObjectNr
      >I;	// 
      BEC;	// 
      L     64;	// 
      >I;	// 
      BEC;	// 
      L     P#146.0;	// --> Pointer  "LineDB1".JobWrite.ObjMask[1]
      L     DBW 20;	// LineDB.VarTemp[1] = ObjectNr
      +I;	// 
      +     -1;	// 
      T     #VarAdrBit;	// --> Address "LineDB1".JobWrite.ObjMask[x]
      AN    DBX [#VarAdrBit];	//  ObjMask[x]
      BEC;	// --> no dymamic data_block
      L     0;	// 
      L     DBW 6;	// "LineDB1".Para.ParAddrObjData
      ==I;	// 
      JC    BSTD;	// 
      SLD   3;	// (Bit-Nr)
      T     #VarBitAdrRead;	// --> BitAddrRead
      L     64;	// 
BLop: T     #VarCountLoop;	// 
      L     0;	// 
      L     DBW [#VarBitAdrRead];	// "LineDB1".ParObjData.ObjXx.ObjNr
      ==I;	// 
      JC    BErr;	// --> error:config. missing
      L     DBW 20;	// LineDB.VarTemp[1] = ObjectNr
      ==I;	// 
      JC    BOK;	// -->  config. found
      L     #VarBitAdrRead;
      +     L#32;
      T     #VarBitAdrRead;
      L     #VarCountLoop;
      LOOP  BLop;
//====Error handling =====================================
BErr: L     12;
      T     DBW 140;	// ->JobRead.ErrCode= error:config.block missing
      L     DBW 20;	// LineDB.VarTemp[1] = ObjectNr
      T     DBW 142;	// ->.JobRead.ErrObject= error:com_err_obj
      BEU;
//=== Return Data ========================================
BOK:  L     #VarBitAdrRead;	// 
      +     L#16;	// 
      T     #VarBitAdrRead;	// 
      L     DBW [#VarBitAdrRead];	// "LineDB1".ParObjData.ObjXx.BytNr
BSTD: T     DBW 22;	// -->"LineDB1".VarTemp[2]= VarDWNr
      BEU;	//  
END:  NOP   0;
NETWORK
TITLE =  Code 2: Subroutine "Reset ObjMask"
//-Rückseten des zum Object n zugehörigen Bit in der Maske 
// LineDB".JobWrite.ObjMask 
// als Quittung, dass das Objekt-Daten ausgewertet wurden
//-Reset the bit of object n in  "LineDB".JobWrite.ObjMask, as answer, that the
// object datas are read.
//
// CALL by methode decoder
// INPUT  : ACTUAL DB BY CALL =L_DB
// INPUT  : LineDB.VarTemp[1] (DBW20) = ObjectNr
//
      L     #CODE;
      L     2;
      <>I;
      JC    BEnd;
      L     0;
      L     DBW 20;	// LineDB.VarTemp[1]= ObjectNr
      >I;
      BEC;
      L     64;
      >I;
      BEC;
      L     DBW 20;	// LineDB.VarTemp[1]= ObjectNr
      +     -1;	// 
      LAR1;
      R     DBX [AR1,P#146.0];	// "LineDB1".JobWrite.ObjMask[x]
      BEU;	// )
BEnd: NOP   0;
NETWORK
TITLE =  Code 3: Send Commmands
//-Befehle von Linie an alle Sektionen verteilen
// als Quittung, dass das Objekt-Daten ausgewertet wurden
//-Send commands from line to all section.
//
// CALL by methode Control and PC Direct Control
// INPUT  : ACTUAL DB BY CALL =Line-DB
// INPUT  : LineDB.VarTemp[7,8] (DBD32): Function
//
      L     #CODE;
      L     3;
      <>I;
      JC    CEnd;
      OPN   DI [DBW 4];	// )-->CALL SECTION-DB[L_DB.ParFirstSecDB]
CLop: L     DBD 32;	//  VarFunction
      L     DID 46;	//  "SecDB".ToASW.Func
      OD;	//  
      T     DID 46;	//  -->"SecDB".ToASW.Func
//- Call next section DB
      L     0;	//  
      L     DIW 8;	//  "SecDB1".Para.ParNextSecDB
      ==I;	//  
      BEC;	//  
      OPN   DI [DIW 8];	// -->CALL SECTION-DB "SecDB1".Para.ParNextSecDB]
      JU    CLop;	// 
CEnd: NOP   0;
NETWORK
TITLE =
END_FUNCTION

